// SIMATIC STEP 7 (V5.x) project ONOFF_D
// program: S7 Program(1)

SYMBOL_TABLE
"ONOFF_DELAY"	FB 138	FB 138
END_SYMBOL_TABLE

FUNCTION_BLOCK "ONOFF_DELAY"	// FB 138
TITLE = Блок задержки отключения
//Введем задержку отключения ПЧ и контактора, при этом включение будем проводить 
//без какой-либо задержки. По хорошему надо сделать блок только включили, чтобы 
//проводить эту проверку, или вообще надо всех смотреть есть ли частота и если 
//она падает до нуля больше чем на время Т все плохо.
AUTHOR : ETSystem
VERSION : 0.0
VAR_INPUT
  ON_OFF : BOOL ;	//Включение, выключение механизма
  T_DEBOUNCE : S5TIME  := S5T#20S;
  TOFF_DELAY : S5TIME  := S5T#10S;	//Задержка времени (S5T)
  F_DELAY_VIKL : REAL  := 1.000000e+000;	//Частота при которой происходит отключение контактора при выключении
  F_DELAY_VKL : REAL  := 2.400000e+001;	//Частота при которой происходит отключение контактора при включении
  FREQ : REAL ;	//Частота на выходе ПЧ
  IN_ALARM1 : BOOL ;	//Авария на входе 1
  IN_ALARM2 : BOOL ;	//Авария на входе 2
  IN_ALARM3 : BOOL ;	//Авария на входе 3
END_VAR
VAR_OUTPUT
  QFC_ONOFF : BOOL ;	//ЧП включен(1)/выключен(0) - Выходная
  QSW_ONOFF : BOOL ;	//Контактор включен(1)/выключен(0) - Выходная
  QFC_ALARM : BOOL ;
END_VAR
VAR
  FC_ONOFF : BOOL ;	//ЧП включен(1)/выключен(0)
  SW_ONOFF : BOOL ;	//Контактор включен(1)/выключен(0)
  FC_ALARM : BOOL ;
END_VAR
BEGIN
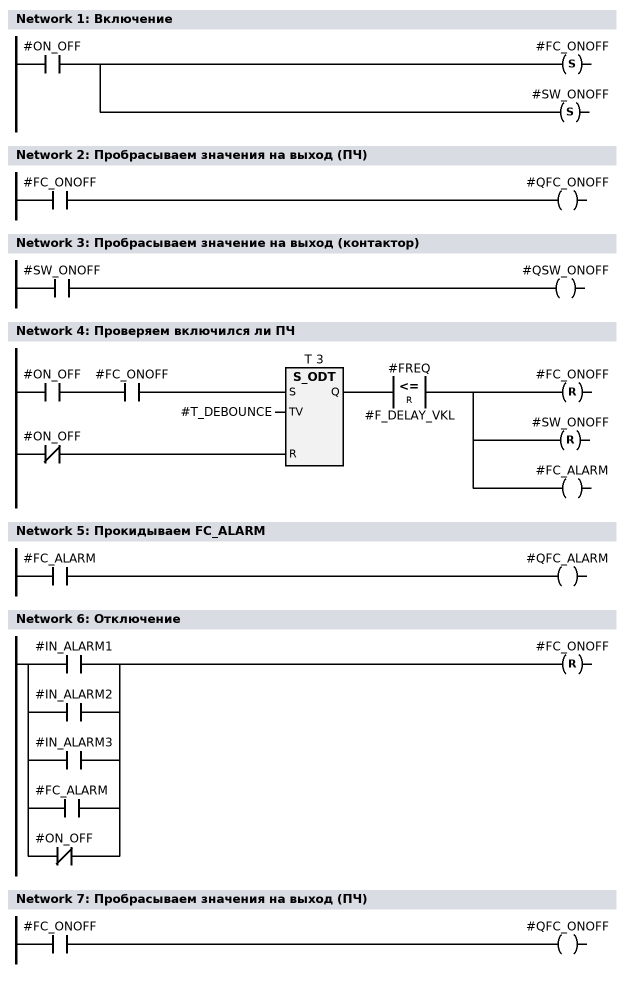
NETWORK
TITLE = Включение
//При наличии сигнала, все включаем, без каких либо задержек
      A     #ON_OFF;
      S     #FC_ONOFF;
      S     #SW_ONOFF;
NETWORK
TITLE = Пробрасываем значения на выход (ПЧ)
      A     #FC_ONOFF;
      =     #QFC_ONOFF;
NETWORK
TITLE = Пробрасываем значение на выход (контактор)
      A     #SW_ONOFF;
      =     #QSW_ONOFF;
NETWORK
TITLE = Проверяем включился ли ПЧ
//Если через время частота не появилась, значит ПЧ не включился и отрубаем все к 
//чертикам. СБРОСА ТАЙМЕРА НЕТ. 
      A(;
      A     #ON_OFF;
      A     #FC_ONOFF;
      L     #T_DEBOUNCE;
      SD    T 3;
      AN    #ON_OFF;
      R     T 3;
      NOP   0;
      NOP   0;
      A     T 3;
      );
      A(;
      L     #FREQ;
      L     #F_DELAY_VKL;
      <=R;
      );
      R     #FC_ONOFF;
      R     #SW_ONOFF;
      =     #FC_ALARM;
NETWORK
TITLE = Прокидываем FC_ALARM
      A     #FC_ALARM;
      =     #QFC_ALARM;
NETWORK
TITLE = Отключение
//Последовательно отключаем ПЧ и контактор, сперва ПЧ(плюс аварии)
      O     #IN_ALARM1;
      O     #IN_ALARM2;
      O     #IN_ALARM3;
      O     #FC_ALARM;
      ON    #ON_OFF;
      R     #FC_ONOFF;
NETWORK
TITLE = Пробрасываем значения на выход (ПЧ)
      A     #FC_ONOFF;
      =     #QFC_ONOFF;
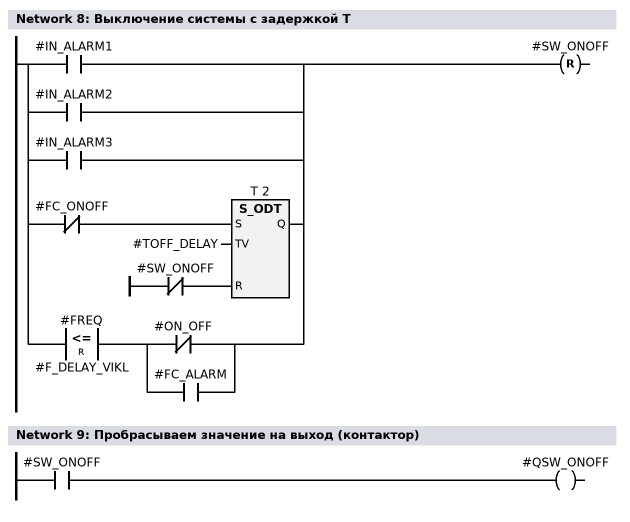
NETWORK
TITLE = Выключение системы с задержкой T
//Затем отключаем контактор, либо по таймеру с задержкой T_DELAY, либо если 
//частота на ПЧ упала ниже F_DELAY, либо авария на входе
      O     #IN_ALARM1;
      O     #IN_ALARM2;
      O     #IN_ALARM3;
      O(;
      AN    #FC_ONOFF;
      L     #TOFF_DELAY;
      SD    T 2;
      AN    #SW_ONOFF;
      R     T 2;
      NOP   0;
      NOP   0;
      A     T 2;
      );
      O;
      A(;
      L     #FREQ;
      L     #F_DELAY_VIKL;
      <=R;
      );
      A(;
      ON    #ON_OFF;
      O     #FC_ALARM;
      );
      R     #SW_ONOFF;
NETWORK
TITLE = Пробрасываем значение на выход (контактор)
      A     #SW_ONOFF;
      =     #QSW_ONOFF;
NETWORK
TITLE = Обработка аварий
END_FUNCTION_BLOCK

ORGANIZATION_BLOCK OB 1
TITLE = "Main Program Sweep (Cycle)"
VERSION : 0.1
VAR_TEMP
  OB1_EV_CLASS : BYTE ;	//Bits 0-3 = 1 (Coming event), Bits 4-7 = 1 (Event class 1)
  OB1_SCAN_1 : BYTE ;	//1 (Cold restart scan 1 of OB 1), 3 (Scan 2-n of OB 1)
  OB1_PRIORITY : BYTE ;	//Priority of OB Execution
  OB1_OB_NUMBR : BYTE ;	//1 (Organization block 1, OB1)
  OB1_RESERVED_1 : BYTE ;	//Reserved for system
  OB1_RESERVED_2 : BYTE ;	//Reserved for system
  OB1_PREV_CYCLE : INT ;	//Cycle time of previous OB1 scan (milliseconds)
  OB1_MIN_CYCLE : INT ;	//Minimum cycle time of OB1 (milliseconds)
  OB1_MAX_CYCLE : INT ;	//Maximum cycle time of OB1 (milliseconds)
  OB1_DATE_TIME : DATE_AND_TIME ;	//Date and time OB1 started
END_VAR
BEGIN
// (block stored without names or comments; labels and parameter names are numbered)
END_ORGANIZATION_BLOCK
